KUKA KRL data list: StiffySense_Test_IMU.dat

&ACCESS RVO1
&COMMENT
DEFDAT StiffySense_Test_IMU PUBLIC

DECL E6AXIS StiffyIMURotate
DECL BOOL StiffyMove
DECL BOOL StiffyPointReceived
DECL E6POS HOME

ENDDAT
